VAR_GLOBAL






END_VAR

(* stored: Version 1.1.0.1, ProductVersion 3.1.4022.12
   GVL GVL_GATT: Id {5818d4b8-e121-409d-b0dc-964a5d06ddad} *)
